FUNCTION_BLOCK CiA_DS402Controlword_Vacon EXTENDS CiA_DS402Controlword
VAR_INPUT
	AlarmReset				:	BOOL; //Manufacturere specific Bit 12 

END_VAR
VAR_OUTPUT
END_VAR
VAR
END_VAR

;

METHOD PUBLIC createControlword : BOOL
VAR_INPUT
	StatusState												: eCiA_DS402_STATUS_STATE;
END_VAR
VAR_IN_OUT
	Controlword												:	UINT;
END_VAR
	
	createControlword									:= SUPER^.createControlword(StatusState,Controlword);
	Controlword.11										:= AlarmReset;	
	
	
(*****************************************************************************)
END_METHOD

END_FUNCTION_BLOCK

(* stored: Version 1.1.0.1, ProductVersion 3.1.4024.13
   POU CiA_DS402Controlword_Vacon: Id {d02ce510-914f-4cac-b1b9-479dfed1a7a7}, SpecialFunc None
   Method createControlword: Id {c9a9f519-efce-464e-b494-2e367d76e912} *)
